INTERFACE I_Syntax_BaseDevice EXTENDS __SYSTEM.IQueryInterface

METHOD M_Start : BOOL
VAR_INPUT
    bForce : BOOL;
END_VAR
END_METHOD

METHOD M_Stop : BOOL
END_METHOD

PROPERTY P_IsRunning : BOOL
GET
END_GET
END_PROPERTY

END_INTERFACE

(* stored: Version 1.1.0.1, ProductVersion 3.1.4024.16
   Itf I_Syntax_BaseDevice: Id {2f268b66-04fb-4e1f-8ed2-37e106521d68}
   Method M_Start: Id {ff38a999-85f8-4aed-bd04-2308ab074300}
   Method M_Stop: Id {84f79bc0-31f7-49b2-b128-e4db0d2d12a1}
   Property P_IsRunning: Id {fc4134dd-42fe-4916-9dba-cdd9547ce85f}
   Get Get: Id {42720f7b-cf68-4c66-83c4-95614aa23c7c} *)
